// TIA Portal project "Project1" (V18)

(* hardware
DEVICE "S7-1200 station_1"  S7-1200 Station
   slot 0: "Rack_0"  S7-1200 Rack  Rack  V1.0
   slot 1: "PLC_1"  CPU 1214C DC/DC/DC  6ES7 214-1AG31-0XB0  V3.0
*)

// ===== PLC "PLC_1"  CPU 1214C DC/DC/DC =====

VAR_GLOBAL   // PLC tag table "Default tag table"
   "En_Read" AT %M2.0 : Bool;
   "Data_Rec_ESP" AT %MW50 : Word;
   "En_Con1" AT %M2.1 : Bool;
   "I00" AT %I0.0 : Bool;
   "Clock_Byte" AT %MB0 : Byte;
   "Clock_10Hz" AT %M0.0 : Bool;
   "Clock_5Hz" AT %M0.1 : Bool;
   "Clock_2.5Hz" AT %M0.2 : Bool;
   "Clock_2Hz" AT %M0.3 : Bool;
   "Clock_1.25Hz" AT %M0.4 : Bool;
   "Clock_1Hz" AT %M0.5 : Bool;
   "Clock_0.625Hz" AT %M0.6 : Bool;
   "Clock_0.5Hz" AT %M0.7 : Bool;
   "System_Byte" AT %MB1 : Byte;
   "FirstScan" AT %M1.0 : Bool;
   "DiagStatusUpdate" AT %M1.1 : Bool;
   "AlwaysTRUE" AT %M1.2 : Bool;
   "AlwaysFALSE" AT %M1.3 : Bool;
   "Data_Send_ESP" AT %MW52 : Word;
   "I15" AT %I1.7 : Bool;
   "I14" AT %I1.6 : Bool;
   "I13" AT %I1.5 : Bool;
   "I12" AT %I1.4 : Bool;
   "I11" AT %I1.3 : Bool;
   "I10" AT %I1.2 : Bool;
   "I09" AT %I1.1 : Bool;
   "I08" AT %I1.0 : Bool;
   "I07" AT %I0.7 : Bool;
   "I06" AT %I0.6 : Bool;
   "I05" AT %I0.5 : Bool;
   "I04" AT %I0.4 : Bool;
   "I03" AT %I0.3 : Bool;
   "I02" AT %I0.2 : Bool;
   "I01" AT %I0.1 : Bool;
   "Tag_1" AT %M2.2 : Bool;
   "AI1" AT %IW64 : Int;
   "Send_DC_PWM" AT %MW70 : Int;
   "Send_Sentido_Horario" AT %M3.2 : Bool;
   "Stop" AT %M3.1 : Bool;
   "Start" AT %M3.0 : Bool;
   "Send_Def_ESP" AT %MW4 : Int;
   "Send_Data_ESP" AT %M3.3 : Bool;
   "MEM_Endereco1" AT %M3.4 : Bool;
   "MEM_motorOn" AT %M3.5 : Bool;
   "MEM_direcao" AT %M3.6 : Bool;
   "MEM_PWM" AT %MW6 : Int;
   "MEM_Endereco2" AT %M3.7 : Bool;
   "MEM_MotorOff" AT %M8.0 : Bool;
END_VAR

// folder: System blocks/Program resources

DATA_BLOCK "PLC_1_Send_DB"   // DB4
{ S7_Optimized_Access := 'TRUE' }
AUTHOR : SIMATIC
FAMILY : MC7Plus
NAME : TCON_Prm
VERSION : 1.0
// stored: InstanceOfName TCON_Param
"TCON_Param"
BEGIN
   ID := 2;
   REM_TSAP_ID_LEN := 0;
   LOCAL_TSAP_ID[1] := B#16#07;
   LOCAL_TSAP_ID[2] := B#16#E7;
   LOCAL_TSAP_ID_LEN := 2;
   ACTIVE_EST := false;
   REM_STADDR[1] := 192;
   REM_STADDR[2] := 168;
   REM_STADDR[4] := 123;
END_DATA_BLOCK

DATA_BLOCK "PLC_1_Receive_DB"   // DB5
{ S7_Optimized_Access := 'TRUE' }
AUTHOR : SIMATIC
FAMILY : MC7Plus
NAME : TCON_Prm
VERSION : 1.0
// stored: InstanceOfName TCON_Param
"TCON_Param"
BEGIN
   ID := 1;
   REM_TSAP_ID_LEN := 0;
   LOCAL_TSAP_ID[1] := B#16#07;
   LOCAL_TSAP_ID[2] := B#16#E8;
   LOCAL_TSAP_ID_LEN := 2;
   ACTIVE_EST := false;
   REM_STADDR[1] := 192;
   REM_STADDR[2] := 168;
   REM_STADDR[4] := 123;
END_DATA_BLOCK

// folder: (top level)

FUNCTION "SendWord" : Void   // FC1, SCL
{ S7_Optimized_Access := 'TRUE' }
VERSION : 0.1
   VAR_TEMP
      tempWord : Word;
      tempvalorpwm : Word;
      tempendereco : Word;
   END_VAR
BEGIN
   // Montar a WORD de envio da ESP (MW52)

   // Limpa a variável temporária
   #tempWord := W#16#0000;

   // Bits 0 a 7 - PWM pra velocidade do motor

   //#tempvalorpwm := INT_TO_WORD(("AI1" * 255) / 27648);  // NormX e ScaleX aqui
   #tempvalorpwm := INT_TO_WORD("Send_DC_PWM");
   #tempvalorpwm := #tempvalorpwm AND w#16#00FF; // Faz um AND com 0...11111111

   #tempWord := #tempWord OR #tempvalorpwm;

   // Bit 8 - Direção

   IF "Send_Sentido_Horario" THEN
       #tempWord := #tempWord OR w#16#0100; //1 0000 0000 de hexa pra binário
   END_IF;

   // Bit 11 - Ligar/Desligar

   IF "Start" AND NOT "Stop" THEN
       #tempWord := #tempWord OR w#16#0800;
   END_IF;

   // Bits 12 a 15 - endereço ESP

   #tempendereco := INT_TO_WORD("Send_Def_ESP") AND W#16#000F;
   #tempendereco := #tempendereco * W#16#1000; //deslocar em 1 0000 0000 0000
   #tempWord := #tempWord OR #tempendereco;

   // Salva o resultado na memória MW52
   "Data_Send_ESP" := #tempWord;
END_FUNCTION

FUNCTION "Controle_Motor" : Void   // FC2, LAD
{ S7_Optimized_Access := 'TRUE' }
VERSION : 0.1
   VAR_TEMP
      Temp_Vel_Norm : Real;
   END_VAR
BEGIN

REGION Network 1: Selecionar ESP
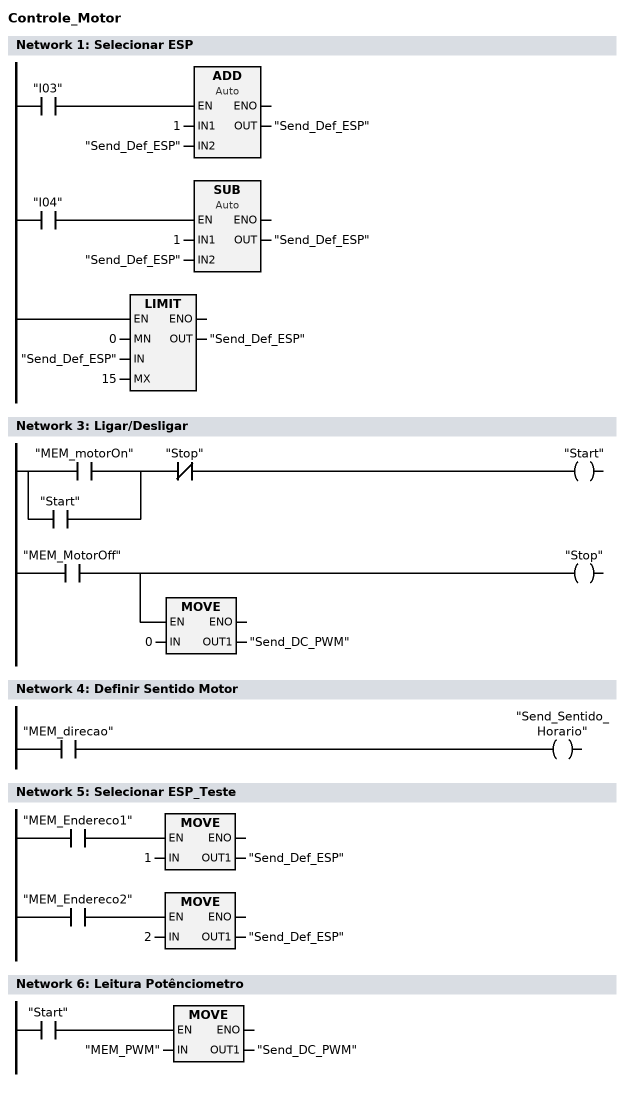
   IF "I03" THEN "Send_Def_ESP" := 1 + "Send_Def_ESP"; END_IF;
   IF "I04" THEN "Send_Def_ESP" := 1 - "Send_Def_ESP"; END_IF;
   "Send_Def_ESP" := LIMIT(MN := 0, IN := "Send_Def_ESP", MX := 15);
END_REGION

REGION Network 3: Ligar/Desligar
   RUNG wire#powerrail
      Contact( "MEM_motorOn" )
      wire#w1
      I_Contact( "Stop" )
      Coil( "Start" )
   END_RUNG
   RUNG wire#powerrail
      Contact( "Start" )
   END_RUNG wire#w1
   RUNG wire#powerrail
      Contact( "MEM_MotorOff" )
      wire#w2
      Coil( "Stop" )
   END_RUNG
   RUNG wire#w2
      { S7_GenerateENO := "TRUE" } Move(in := 0, out1 => "Send_DC_PWM")
   END_RUNG
   // the same network as SCL:
   "Start" := ("MEM_motorOn" OR "Start") AND NOT "Stop";
   "Stop" := "MEM_MotorOff";
   IF "MEM_MotorOff" THEN "Send_DC_PWM" := 0; END_IF;
END_REGION

REGION Network 4: Definir Sentido Motor
   RUNG wire#powerrail
      Contact( "MEM_direcao" )
      Coil( "Send_Sentido_Horario" )
   END_RUNG
   // the same network as SCL:
   "Send_Sentido_Horario" := "MEM_direcao";
END_REGION

REGION Network 5: Selecionar ESP_Teste
   RUNG wire#powerrail
      Contact( "MEM_Endereco1" )
      { S7_GenerateENO := "TRUE" } Move(in := 1, out1 => "Send_Def_ESP")
   END_RUNG
   RUNG wire#powerrail
      Contact( "MEM_Endereco2" )
      { S7_GenerateENO := "TRUE" } Move(in := 2, out1 => "Send_Def_ESP")
   END_RUNG
   // the same network as SCL:
   IF "MEM_Endereco1" THEN "Send_Def_ESP" := 1; END_IF;
   IF "MEM_Endereco2" THEN "Send_Def_ESP" := 2; END_IF;
END_REGION

REGION Network 6: Leitura Potênciometro
   RUNG wire#powerrail
      Contact( "Start" )
      { S7_GenerateENO := "TRUE" } Move(in := "MEM_PWM", out1 => "Send_DC_PWM")
   END_RUNG
   // the same network as SCL:
   IF "Start" THEN "Send_DC_PWM" := "MEM_PWM"; END_IF;
END_REGION
END_FUNCTION

ORGANIZATION_BLOCK "Main"   // OB1, LAD, ProgramCycle
TITLE = "Main Program Sweep (Cycle)"
{ S7_Optimized_Access := 'TRUE' }
VERSION : 0.1
BEGIN

REGION Network 1
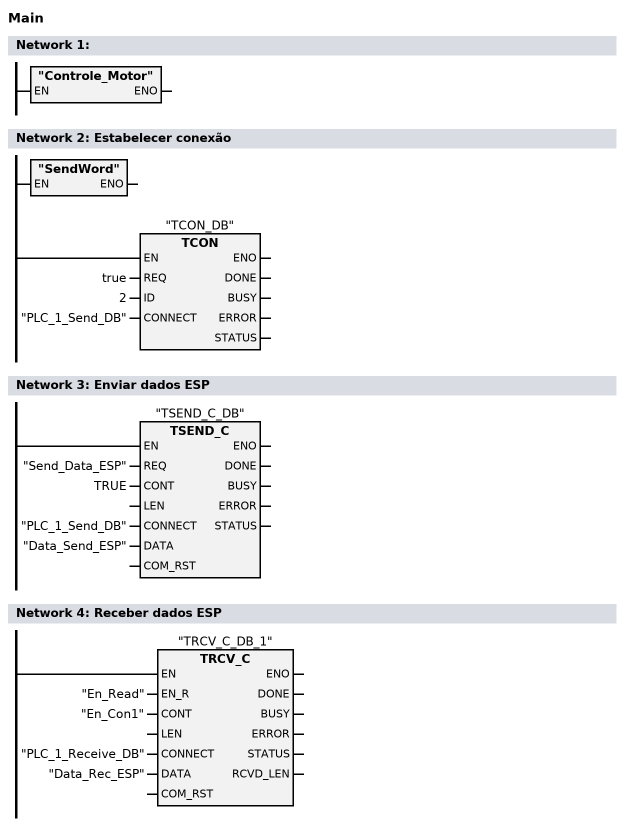
   RUNG wire#powerrail
      "Controle_Motor"()
   END_RUNG
   // the same network as SCL:
   "Controle_Motor"();
END_REGION

REGION Network 2: Estabelecer conexão
   "SendWord"();
   "TCON_DB"(REQ := true, ID := 2, CONNECT := "PLC_1_Send_DB");   // TCON
END_REGION

REGION Network 3: Enviar dados ESP
   "TSEND_C_DB"(REQ := "Send_Data_ESP", CONT := TRUE, CONNECT := "PLC_1_Send_DB", DATA := "Data_Send_ESP");   // TSEND_C
END_REGION

REGION Network 4: Receber dados ESP
   "TRCV_C_DB_1"(EN_R := "En_Read", CONT := "En_Con1", CONNECT := "PLC_1_Receive_DB", DATA := "Data_Rec_ESP");   // TRCV_C
END_REGION
END_ORGANIZATION_BLOCK